{attribute 'Tc2GvlVarNames'}
{attribute 'strict'}
//Tipologia Di Presa dell' Elemento da parte dell'End Effector
TYPE e_Tipo_PresaEndEffector :
(
	TPICK_NOT_DEFINED							:= -1,      (* Tipo di prelievo indefinito *)
	TPICK_PACK									:= 0,		(* Identifica la presa di tipo PACCO *)
	TPICK_PALLET								:= 1,		(* Identifica la presa di tipo PALLET *)
	TPICK_LAYER									:= 2,		(* Identifica la presa di tipo FALDA (CLASSICA A VENTOSE,uitlizzata nel pal. pacchi) *)
	TPICK_LASTRA								:= 3,		(* Identifica la presa di tipo LASTRA (CLASSICA A VENTOSE) *)
	
	
	
	(* Tipologia di presa della falda *)
	TPICK_LAY_VENTOSE							:= 4,		(* Identifica la presa di tipo FALDA A VENTOSE, utilizzata nel pal. Lastre *)
	TPICK_LAY_ARPIONI							:= 5,		(* Identifica la presa di tipo FALDA CON ARPIONI, utilizzata nel pal. Lastre per il polistirolo *)
	
	TPICK_QUADROTTA								:= 10		(* Identifica la presa di tipo LASTRA (CLASSICA A VENTOSE) *)

	//TPICK_UNDEFINED								 := 99     
);
END_TYPE
//  TPICK_NOT_DEFINED = '-1'

(* stored: Version 1.1.0.1, ProductVersion 3.1.4024.11
   EnumerationTextList e_Tipo_PresaEndEffector: Id {c7919730-0437-43f1-ba63-8566b7564986} *)
